(* CODESYS project Monarco HAT library for codesys 0.9.0.3.library
   Author: Aliazzz
   LibDocContent: CommentsAndDocs
   Description: .. _description: 
      
      Library containing device support for Monarco HAT hardware developped by the guys from Monarco.io.
      
      I decided to write this library because the hardware is very solid, but a CODESYS implementation was missing.
      Writing this library was fun, but took a lot of sweat and time, please refer to this work when you use it =).
      
      I am not affiliated with Monarco.io in any way, shape or form.
      
      Released under Unlicense.
      
      
      Enjoy!
      
      
      **Getting started**
      
      To use the HAT, RS-485 and the Realtime Clock under CODESYS, please follow these steps. RTC requires no Linux side config apart from the overlay;
      
      1) On your Raspberry Pi, switch to root user: sudo -s
      
      2) Disable Linux console on UART: **sed 's/ console=serial0,[0-9]\+//' -i /boot/cmdline.txt**
      
      3) Run the following command to get device-tree overlay definition for the RS-485 on the Monarco HAT: **wget www.monarco.io/download/monarco-fix-4-9.dtbo**
      
      4) Copy it to /boot/overlays: **sudo cp monarco-fix-4-9.dtbo /boot/overlays**
      
      5) Afterwards add dtoverlay=monarco-fix-4-9 line to the /boot/config.txt file: **echo dtoverlay=monarco-fix-4-9 >> /boot/config.txt**
      
      6) Reboot your Raspberry Pi: **reboot**
      
      7) After reboot, check the output of the following command: **ls -l /dev/serial0**
      
      8) The response should read **"/dev/serial0 -> ttyAMA0"**
      
      9) Again, switch to root user: **sudo -s  cd etc/**
      
      10) Then: **nano CODESYSControl.cfg**
      
      11) Add the following lines: **[SysCom] Linux.Devicefile=/dev/ttyAMA**
      
      12) Then reboot your Raspberry Pi again: **reboot**
      
      13) After reboot: **Now you can use the HAT, RS-485 and the Real-Time Clock in CODESYS!** from within an IEC application via a comlib of you own flavour (like CAA SerialCOM library).
      
      .. image:: ../Images/MonarcoHAT.png
      
      
      * Real Time Clock (RTC)
      * RS-485 Interface
      * 1-Wire Interface (1w)
      * 4 Digital Inputs
      * 4 Digital Outputs
      * 2 Analog Inputs 12 bits without sign: (0 - 4095) 0..10V / 0..25mA
      * 2 Analog Outputs 12 bit without sign: (0 - 4095) 0..10V
      * LEDs: 1 × orange, 8 × green LEDs
      * Power supply: 10-30 VDC, powers also the Raspberry Pi
      
      
      This library is based on Hardware version 0106, Firmware version 2006.
   Title: Monarco HAT library for Codesys
   Version: 0.9.0.3
   DefaultNamespace: MNR
   DocFormat: reStructuredText
   Company: Monarco.io

Project tree, tasks and I/O mapping:
  libraries: IoDrvGPIO, 3.5.11.0 (3S - Smart Software Solutions GmbH); Raspberry Pi Peripherals, 3.5.11.0 (3S - Smart Software Solutions GmbH); IoStandard, * (System); CAA Memory, * (CAA Technical Workgroup); Standard, * (System); CAA Real Time Clock Extern, * (CAA Technical Workgroup); CAA SerialCom, * (CAA Technical Workgroup)
  function block Monarco_FB [ST]: AfterReadInputs, BeforeWriteOutputs, Initialize, flush, checkCRC, dataTransfer, getCRC, writeRaw, getHATinfo, RS485Baudrate, RS485Mode, HostBaudrate, RS485RxC, RS485TxC, RS485FxC, RS485PxC, setDOut, ServiceRequest, getCpuID, getFwVersion, getHwVersion, getStatus, HWConfig1, Watchdog, getServiceResponse, ControlByte, getDIn, getAIn, setRawTxBuf, getRawRxBuf, setAOut, Counter1Config, Counter2Config, setPWM1freq, setPWM2freq, setDutyCycleDOut1, setDutyCycleDOut2, setDutyCycleDOut3, setDutyCycleDOut4, SetUserLED
  00000000-0000-0000-0000-000000000000|C:\Users\user\Desktop\Monarco HAT\Dev\images\schematics.png
  Library Information/
    function GetLibVersionNumber [ST]
    function GetLibVersion [ST]
    function IsLibReleased [ST]
  Images/
    schematics
    MonarcoHAT
  00000000-0000-0000-0000-000000000000|C:\Users\user\Desktop\Monarco HAT\Dev\images\MonarcoHAT.png
  Datatypes/
    RS485/
      data type stRS485Mode
      data type eRS485Parity
      data type eRS485Databits
      data type eRS485Stopbits
    AIn/
      data type stAIn
    AOut/
      data type stAOut
    DIn/
      data type stDIn
    DOut/
      data type stDOut
    Service/
      data type stServiceRequest
      data type eMonarcoOperation
      data type stMonarcoStatus
      data type eMonarcoComStatus
      data type stMonarcoCmd
      data type stHWConfig1
      data type stControlByte
      data type stHATinfo
      data type eServiceCommand
      data type stServiceResponse
    Counter/
      data type stCounter1Config
      data type eCounterMode
      data type eCounterDirection
      data type eCounterActiveEdge
      data type stCounter2Config
      data type eCounterCapture
    PWM/
      data type ePrescaler
      data type stPWM2
      data type stPWM1
  global variables ParamList
  Functions/
    function getDC [ST]
*)

// Datatypes/Service/stServiceRequest
// Service Request and Service Response structure
// **Setting "Error" is only valid in a Service Response**
TYPE stServiceRequest :
STRUCT
	wServiceValue 	: WORD;
	wServiceAddress : WORD;
/// Error to be examined on a response only! 
/// If set, the response ServiceValue contains one of the following error codes;
///
/// - Invalid adress (code 16#FFFF)
/// 
/// - CRC error (16#CCCC)
///
	xError			: BOOL; 	
END_STRUCT
END_TYPE

// Datatypes/Service/eMonarcoOperation
/// Execution commands for the Monarco HAT via classic command interface
{attribute 'qualified_only'}
{attribute 'strict'}
TYPE eMonarcoOperation :
(
/// Write an entire raw self defined message according to input 
	WriteRaw			:= 0,
/// Write the controlbyte according to input  	
	WriteCtrlByte		:= 1,
/// Write the leds according to input  	
	WriteUserLeds		:= 2,
/// Write Digital Outs according to input	
	WriteDOut			:= 3,
/// Write Analog Outs according to input	
	WriteAOut			:= 4,
/// Write PWM1 frequency according to input	
	WritePWM1Freq		:= 5,
/// Write PWM2 frequency according to input	
	WritePWM2Freq		:= 6,
/// Write Counter1 according to input	
	WriteCNT1			:= 7,
/// Write Counter2 according to input	
	WriteCNT2			:= 8,
/// Write PWM1 duty cycle according to input	
	WriteDutyCycleDOut1	:= 9,
/// Write PWM1 duty cycle according to input	
	WriteDutyCycleDOut2	:= 10,
/// Write PWM1 duty cycle according to input	
	WriteDutyCycleDOut3	:= 11,
/// Write PWM2 duty cycle according to input	
	WriteDutyCycleDOut4	:= 12
) UINT;
END_TYPE

// Datatypes/Service/stMonarcoStatus
/// Monarco HAT Classic Status Structure
{attribute 'qualified_only'}
{attribute 'strict'}
TYPE stMonarcoStatus :
STRUCT
/// Is the Monarco HAT operational?
	xOperational			: BOOL;
/// Operation Command was successfully finished 			 	
	xDone					: BOOL;
/// An errror occuried, see ComStatus			 	
	xError					: BOOL;
/// Has to examined in conjunction with xExecute, xDone and xError				 	
	eComStatus				: eMonarcoComStatus;
/// Controlbyte status 	
	stControlByte			: stControlByte; 
/// Contains most recent service response	
	stLastServiceResponse	: stServiceResponse;
/// User Leds On Off status;
	byUserLeds				:BYTE;
/// Current state of digital In channel values  	
	stDIn					: stDIn;
/// copy of digital Out channel values				
	stDOut					: stDOut;
/// Current state of analog In channel values  				
	stAIn					: stAIn;
/// copy of analog Out channel values
	stAOut					: stAOut;
/// current watchdog time: 100 = 100msec
	uiWatchDog				: UINT;
/// current Baudrate: 300 = 300Bd				
	uiRS485Baudrate			: UINT;
/// Current RS485 communication settings mode				
	stRS485Mode				: stRS485Mode;
/// Current settings for RS485 termination and AI voltage or current-loop mode			
	stHWConfig1 			: stHWConfig1;
/// Current Counter 1 configuration  			
	stCounter1Config		: stCounter1Config;
/// Current Counter 2 configuration	
	stCounter2Config		: stCounter2Config;
/// PWM1 Settings
	stPWM1					: stPWM1;
/// PWM2 Setting
	stPWM2					: stPWM2;
/// Static HAT information like FW version, HW version and CPU ID 	
	stHATinfo				: stHATinfo;
/// RAW receive buffer			
	abyRawRxBuffer			: ARRAY [0..(ParamList.MONARCO_STRUCT_SIZE-1)] OF BYTE; 
END_STRUCT
END_TYPE

// Datatypes/Service/eMonarcoComStatus
/// Monarco HAT Communication Status
{attribute 'qualified_only'}
{attribute 'strict'}
TYPE eMonarcoComStatus :
(	
/// Succes: Rx/Tx sent succesfully
	Succes			 		:= 0,
/// Error: Rx/Tx fail
	Error					:= 1,
/// Device not found on the bus
	SPIdeviceNotFound		:= 2,
/// No commands are currently executed. Is xExecute command on the Function Block set?
	SPIidleNoExecute		:= 3,
/// The received message was crippled and dropped
	CrcFail 				:= 4 
) UINT;
END_TYPE

// Datatypes/Service/stMonarcoCmd
/// Monarco Classic Command Structure
{attribute 'qualified_only'}
{attribute 'strict'}
TYPE stMonarcoCmd :
STRUCT
/// Starts a single operation of type "eFunction" on a rising edge of xExecute
	xExecute			: BOOL;	
/// Command to be executed on rising edge of "xExecute"			
	eOperation			: eMonarcoOperation;
/// Use in combination with "eOperation.WRITE_RAW". Setting a CRC is not neccesary, it will be calculated and added automatically	
	abyTxBuffer			: ARRAY [0..(ParamList.MONARCO_STRUCT_SIZE-1)] OF BYTE;
/// For use in combination with "eOperation.WRITE_CTRLBYTE"
	stControlByte		: stControlByte;
/// For use in combination with "eOperation.WRITE_USERLEDS"
	byLeds				: BYTE;
/// For use in combination with "eOperation.WRITE_DOut"		
	stDOut				: stDOUT;
/// For use in combination with "eOperation.WRITE_AOut"			
	stAOut				: stAOut;
/// For use in combination with "eOperation.WRITE_Counter1"			
	stCounter1			: stCounter1Config;
/// For use in combination with "eOperation.WRITE_Counter2"
	stCounter2			: stCounter2Config;
/// For use in combination with "eOperation.WRITE_PWM1Frequency" 
	PWM1freq			: UDINT;
/// For use in combination with "eOperation.WRITE_PWM2Frequency" 
	PWM2freq			: UDINT;
/// For use in combination with "eOperation.WRITE_DutyCycleDOut1" 
	rDutyCycleDOut1		: REAL;
/// For use in combination with "eOperation.WRITE_DutyCycleDOut1" 
	rDutyCycleDOut2		: REAL;
/// For use in combination with "eOperation.WRITE_DutyCycleDOut1" 
	rDutyCycleDOut3		: REAL;
/// For use in combination with "eOperation.WRITE_DutyCycleDOut1" 
	rDutyCycleDOut4		: REAL;
END_STRUCT
END_TYPE

// Datatypes/Service/stHWConfig1
/// Set AnalogIn Channels to Voltage or Current Loop mode,
/// Set RS-485 termination resistor
TYPE stHWConfig1 :
STRUCT
/// AIN1 current loop shunt resistor enable (TRUE / FALSE)
    xAIn1shunt  	: BOOL; 
/// AIN2 current loop shunt resistor enable (TRUE / FALSE)
    xAIn2shunt  	: BOOL;
/// RS-485 termination resistor enable (TRUE / FALSE)
	xTerminated		: BOOL;	
END_STRUCT
END_TYPE

// Datatypes/AOut/stAOut
/// Analog Outputs
TYPE stAOut :
STRUCT
	/// 0..4095 = 0..10V
	wAOut1			: WORD;
	/// 0..4095 = 0..10V
	wAOut2			: WORD; 
END_STRUCT
END_TYPE

// Datatypes/Service/stControlByte
TYPE stControlByte :
STRUCT
/// Status LED mask
/// set 1 for control LED0 by Control byte / Status LED on
/// set 0 for default LED0 function (system status indication, see Monarco HAT Hardware Reference Manual)
	xStatusLedCtrl		: BOOL;
/// Status LED on 
/// Set 1 for LED0 lit on 
/// Set 0 for LED0 off: only applicable if Control byte / Status LED mask set 1
	xStatusLedValue		: BOOL;
/// 1-Wire power shutdown 
/// Set 1 for 1-Wire bus power down (useful for bus reset in case of freeze) 
/// Set 0 for normal operation
	xOneWireShutdown	: BOOL;
/// RESERVED - allways set 0
	xReserved 			: BOOL := FALSE;
/// Counter 1 reset 
/// Set 1 for COUNTER1 Value reset request
/// Set 0 for normal operation. 
/// Reset operation is edge-triggered and its completion is signalised by Statusbyte/Counter 1/2 reset done bit
	xCounter1Reset		: BOOL;
/// Counter 2 reset 
/// Set 1 for COUNTER2 Value reset request
/// Set 0 for normal operation. 
/// Reset operation is edge-triggered and its completion is signalised by Statusbyte/Counter 1/2 reset done bit
	xCounter2Reset		: BOOL;
/// [FUTURE] Sign of Life 0/1 - should be incremented with each data transfer as 2bit number low/high bit, used by firmware as health check of SPI Master
	xSignOfLife0		: BOOL;
/// [FUTURE] Sign of Life 0/1 - should be incremented with each data transfer as 2bit number low/high bit, used by firmware as health check of SPI Master
	xSignOfLife1		: BOOL; 
END_STRUCT
END_TYPE

// Datatypes/DIn/stDIn
/// Digital Inputs
TYPE stDIn :
STRUCT
	xDIn1			: BOOL;
	xDIn2			: BOOL;
	xDIn3			: BOOL;
	xDIn4			: BOOL;
END_STRUCT
END_TYPE

// Datatypes/Service/stHATinfo
/// Returns Firmware, Hardware and CPU revision
TYPE stHATinfo :
STRUCT
/// Monarco HAT Firmware Version
	dwFwVersion			: DWORD;
/// Monarco HAT Hardware Version 
	dwHwversion			: DWORD;
/// Monarco HAT MCU CPU ID
	lwCpuID				: LWORD;
END_STRUCT
END_TYPE

// Datatypes/AIn/stAIn
/// Analog Inputs
TYPE stAIn :
STRUCT
	/// 0..4095 equals 0..10V or 0..25mA, see stHWConfig1_
	wAIn1			: WORD;
	/// 0..4095 equals 0..10V or 0..25mA, see stHWConfig1_
	wAIn2			: WORD;
END_STRUCT
END_TYPE

// Datatypes/DOut/stDOut
/// Digital Outputs
TYPE stDOut :
STRUCT
	xDOut1				: BOOL;
	xDOut2				: BOOL; 
	xDOut3				: BOOL;
	xDOut4				: BOOL; 
END_STRUCT
END_TYPE

// Datatypes/Service/eServiceCommand
/// Registers are Read-only [R], Read-Write [RW] or Write-only [W].
{attribute 'qualified_only'}
{attribute 'strict'}
TYPE eServiceCommand  :
(
/// Read: 0xABCD = OK, [FUTURE] "watchdog triggered", 
/// Write [FUTURE]: - accept only 0xABCD = reset status
	SDC_FIXED_STATUSWORD := 16#0000,
/// Firmware Version - Low Word [R] 
	SDC_FIXED_FWVERL	 := 16#0001,
/// Firmware Version - High Word [R] 
	SDC_FIXED_FWVERH	 := 16#0002,
/// Hardware Version - Low Word [R]
	SDC_FIXED_HWVERL	 := 16#0003,
/// Hardware Version - High Word [R]
	SDC_FIXED_HWVERH	 := 16#0004,
/// MCU Unique ID 1 [R]
	SDC_FIXED_CPUID1	 := 16#0005, 
/// MCU Unique ID 2 [R]
	SDC_FIXED_CPUID2	 := 16#0006, 
/// MCU Unique ID 3 [R]
	SDC_FIXED_CPUID3	 := 16#0007,
/// MCU Unique ID 4 [R]
	SDC_FIXED_CPUID4	 := 16#0008, 
/// HW Config 1 [RW]
/// 
/// * bit 00 - RS-485 termination resistor enable
/// 
/// * bit 01 - AIN1 current loop shunt resistor enable
///  
/// * bit 02 - AIN2 current loop shunt resistor enable
/// 
/// * bit 03..15 - RESERVED (write zeros)
	SDC_FIXED_HWConfig1  := 16#000A,
/// Watchdog Timeout [RW]
/// 
/// Unit: 1 ms; 0 = watchdog disabled; default = 100
	SDC_FIXED_WATCHDOG	 := 16#000F, 
/// HAT RS-485 Baudrate [RW]
///  
/// Unit: 100 Bd, Min: 3 (300 Bd), Max 10000 (1 MBd)
	SDC_FIXED_RS485BAUD  := 16#0010, 
/// HAT RS-485 Mode [RW]
/// 
/// * bit 00..02 - parity - 0: none, 1: even, 2: odd;
/// 
/// * bit 03..04 - data bits: 0: 5, 1: 6, 2: 7, 3: 8; 
/// 
/// * bit 05..06 - stop bits: 0: half, 1: one, 2: one and half, 3: two; 
/// 
/// * bit 07..15 - RESERVED (write zeros)
	SDC_FIXED_RS485MODE  := 16#0011,
/// Host (Pi) UART Baudrate [RW] Unit: 100 Bd, Min: 3 (300 Bd), Max 10000 (1 MBd); 
/// 
/// set to 0 to disable Host UART (set Monarco pins to Hi-Z) when you are using it for another external device.
	SDC_FIXED_HOST_UART  := 16#0012,
/// RS-485 Bytes Received Diagnostics Counter [R]
	SDC_FIXED_RS485_RxC	 := 16#0014,
/// RS-485 Bytes Transmitted Diagnostics Counter [R]
    SDC_FIXED_RS485_TxC  := 16#0015,
/// RS-485 RX Framing Error Diagnostics Counter [R]
    SDC_FIXED_RS485_FxC	 := 16#0018,
/// RS-485 RX Parity Error Diagnostics Counter [R]
    SDC_FIXED_RS485_PxC  := 16#0019,
/// COUNTER1 Configuration [W]
/// 
/// * bit 00..02 - mode: 0: off, 1: pulse counting, 2: quadrature encoder,
/// 
/// * bit 03..05 - direction (only for pulse counting mode): 0: up, 1: [FUTURE] external control, low/high = up/down,
/// 
/// * bit 06..07 - active edge (only for pulse counting mode): 0: rising, 1: falling, 2: both,
/// 
/// * bit 08..15 - RESERVED (write zeros)
	SDC_FIXED_CNT1MODE 	 := 16#0024, 
/// COUNTER2 Configuration [W]
/// 
/// * bit 00..02 - mode: 0: off, 1: pulse counting, 2: quadrature encoder,
/// 
/// * bit 03..05 - direction (only for pulse counting mode): 0: up, 1: [FUTURE] external control, low/high = up/down,
/// 
/// * bit 06..07 - active edge (only for pulse counting mode): 0: rising, 1: falling, 2: both,
/// 
/// * bit 08..09 - CAPTURE function active edge: 0: disabled, 2: [FUTURE] falling, 3: [FUTURE] both,
/// 
/// * bit 10..15 - RESERVED (write zeros)
	SDC_FIXED_CNT2MODE	 := 16#0025,
/// PERSISTENT [FUTURE] parameters area (64 registers, 128 BYTE) 
/// Now for manufacturer use only.
	SDC_PERSISTENT_MIN 	 := 16#0F00,
/// PERSISTENT [FUTURE] parameters area (64 registers, 128 BYTE) 
/// Now for manufacturer use only. 
	SDC_PERSISTENT_MAX 	 := 16#0F3F  
) UINT;
END_TYPE

// Datatypes/RS485/stRS485Mode
/// Monarco HAT RS485 UART settings
TYPE stRS485Mode :
STRUCT
	eParity		 : eRS485Parity;
	eDatabits	 : eRS485Databits;
	eStopbits	 : eRS485Stopbits;
END_STRUCT
END_TYPE

// Datatypes/RS485/eRS485Parity
{attribute 'qualified_only'}
{attribute 'strict'}
TYPE eRS485Parity :
(
	None := 0, 	/// No parity check
	Even := 1,	/// Even parity check
 	Odd  := 2	/// Odd parity check
) UINT;
END_TYPE

// Datatypes/RS485/eRS485Databits
{attribute 'qualified_only'}
{attribute 'strict'}
TYPE eRS485Databits :
(
	Five 	:= 0,	// 1 Byte contains 5 databits
	Six 	:= 1,	// 1 Byte contains 6 databits
	Seven 	:= 2,	// 1 Byte contains 7 databits
	Eight 	:= 3	// 1 Byte contains 8 databits
) UINT;
END_TYPE

// Datatypes/RS485/eRS485Stopbits
{attribute 'qualified_only'}
{attribute 'strict'}
TYPE eRS485Stopbits :
(
	Half 		:= 0,	// 1/2 stopbit
	One 		:= 1,	// 1 stopbit
	OneAndAHalf := 2,	// 1-1/2 stopbits
	Two 		:= 3	// 2 stopbits
) UINT;
END_TYPE

// Datatypes/Service/stServiceResponse
// Alias of Service Request
TYPE stServiceResponse : stServiceRequest; 
END_TYPE

// Datatypes/Counter/stCounter1Config
/// COUNTER1 Configuration;
///   Mode;
///	   * Off,
///    * Pulse counting,
///    * Quadrature encoder,
///   Direction (only for pulse counting mode):
///     * Up
///     * [FUTURE] external control, low/high = up/down
///   Active Edge (only for pulse counting mode):
///     * Rising
///     * Falling
///     * Both
TYPE stCounter1Config :
STRUCT
	eMode		: eCounterMode;
	eDirection	: eCounterDirection;
	eActiveEdge	: eCounterActiveEdge;
END_STRUCT
END_TYPE

// Datatypes/Counter/eCounterMode
{attribute 'qualified_only'}
{attribute 'strict'}
TYPE eCounterMode :
(
	Off 				:= 0,
	PulseCounting		:= 1,
	QuadratureEncoder	:= 2
) UINT;
END_TYPE

// Datatypes/Counter/eCounterDirection
{attribute 'qualified_only'}
{attribute 'strict'}
TYPE eCounterDirection :
(
	Up					:= 0,
	External_Control1	:= 1 //[FUTURE] external control, low/high = up/down
) UINT;
END_TYPE

// Datatypes/Counter/eCounterActiveEdge
{attribute 'qualified_only'}
{attribute 'strict'}
TYPE eCounterActiveEdge :
(
	Rising	:= 0,
	Falling	:= 1,
	Both	:= 2
) UINT;
END_TYPE

// Datatypes/Counter/stCounter2Config
/// COUNTER2 Configuration;
///   Mode;
///	   * Off,
///    * Pulse counting,
///    * Quadrature encoder,
///   Direction (only for pulse counting mode):
///     * Up
///     * [FUTURE] external control, low/high = up/down
///   Active Edge (only for pulse counting mode):
///     * Rising
///     * Falling
///     * Both
///   CAPTURE function active edge:
///     * Disabled
///     * [FUTURE] rising
///     * [FUTURE] falling
///     * [FUTURE] both
TYPE stCounter2Config : 
STRUCT
	Mode		: eCounterMode;
	Direction	: eCounterDirection;
	ActiveEdge	: eCounterActiveEdge;
	Capture		: eCounterCapture;
END_STRUCT
END_TYPE;

// Datatypes/Counter/eCounterCapture
{attribute 'qualified_only'}
{attribute 'strict'}
TYPE eCounterCapture :
(
	Disabled 	:= 0,
	Rising 		:= 1, // [FUTURE]
	Falling 	:= 2, // [FUTURE]
	Both		:= 3  // [FUTURE]
) UINT;
END_TYPE

// Datatypes/PWM/ePrescaler
{attribute 'qualified_only'}
{attribute 'strict'}
TYPE ePrescaler :
(	
	ScaleFactor1	:= 0,	/// PWM Prescale factor is set to 1
	ScaleFactor8 	:= 1,	/// PWM Prescale factor is set to 8
	ScaleFactor64 	:= 2,	/// PWM Prescale factor is set to 64
	ScaleFactor512 	:= 3	/// PWM Prescale factor is set to 512
) UDINT;
END_TYPE

// Datatypes/PWM/stPWM2
TYPE stPWM2 :
STRUCT
	/// period of PWM2 Ch A (DOut4)	(Hz)
	Freq			: UDINT;
	/// Duty Cycle of PWM2 Ch A (DOut4)	
	DutyCycleDOut4	: REAL;
END_STRUCT
END_TYPE

// Datatypes/PWM/stPWM1
TYPE stPWM1 :
STRUCT
	/// period of PWM1 Ch A, B and C (DOut1, 2 and 3) (Hz)
	Freq			: UDINT;
	/// Duty Cycle of PWM1 Ch A (DOut1)	
	DutyCycleDOut1	: REAL;
	/// Duty Cycle of PWM1 Ch B (DOut2)	
	DutyCycleDOut2	: REAL;
	/// Duty Cycle of PWM1 Ch C (DOut3)	
	DutyCycleDOut3	: REAL;
END_STRUCT
END_TYPE

// ParamList
{attribute 'qualified_only'}
VAR_GLOBAL CONSTANT
	MONARCO_STRUCT_SIZE 				: UINT := 26;	
	MONARCO_SERVICE_STATUS_OK 			: WORD := 16#ABCD;
	MONARCO_SERVICE_ERROR_UNKNOWN_REG 	: WORD := 16#FFFF;
	MONARCO_SERVICE_ERROR_CRC 			: WORD := 16#CCCC;
	SDC_ADDRESS_MASK					: WORD := 16#0FFF;		                            
	MONARCO_ADC_RANGE_MAX 				: WORD := 16#4095;
END_VAR

// Monarco_FB
FUNCTION_BLOCK Monarco_FB EXTENDS SPI
VAR_INPUT
	Cmd						: stMonarcoCmd;
END_VAR
VAR_OUTPUT
	Status					: stMonarcoStatus;
END_VAR
VAR
	uiNumberOfDevices		: UINT;		/// Beware, this Library does **NOT** support implementation of multiple SPI devices!
	xGetInitialStatusInfo	: BOOL;		/// Get status info on startup once
	fbR_TRIG				: R_TRIG;	/// FB internal rising edge trigger for xExecute input
	abyIntTxBuf				: ARRAY [0..(ParamList.MONARCO_STRUCT_SIZE-1)] OF BYTE;  
	abyIntRxBuf				: ARRAY [0..(ParamList.MONARCO_STRUCT_SIZE-1)] OF BYTE;  
END_VAR

//********************************
//	base SPI implementation 
//********************************
SUPER^();


//********************************
//		get SPI State 
//********************************
CASE _iState OF
0:
	IF SUPER^.init() THEN
		_iState := 1;
	END_IF	

1:	
	_iState := 10;
	xGetInitialStatusInfo := TRUE;
END_CASE


//********************************
//		is device operational 
//********************************
IF _iState = 10 THEN
	Status.xOperational		:=	TRUE;
ELSE
	Status.xOperational		:=	FALSE;
END_IF


//********************************
// Get Initial startup Status Info 
//******************************** 
IF xGetInitialStatusInfo THEN
	THIS^.getHATinfo();				// all property calls are done via status.gthatinfo to reduce SPI bandwidth on ponintless static info.
	THIS^.Status.stControlByte		:= THIS^.ControlByte;	
	THIS^.Status.stHWConfig1		:= THIS^.HWConfig1;
	THIS^.Status.uiRS485Baudrate	:= THIS^.RS485Baudrate;
	THIS^.Status.stRS485Mode	 	:= THIS^.RS485Mode;
	THIS^.Status.uiWatchDog		 	:= THIS^.Watchdog;
	THIS^.Status.stCounter1Config	:= THIS^.Counter1Config;
	THIS^.Status.stCounter2Config	:= THIS^.Counter2Config;	
	xGetInitialStatusInfo 			:= FALSE;
END_IF


//********************************
//		Operation Mode
//********************************
// No execute, set feedback to inform user
IF NOT Cmd.xExecute THEN				
	Status.xError			:=	FALSE;
	Status.xDone			:=  FALSE;
	Status.eComStatus		:= 	eMonarcoComStatus.SPIIdleNoExecute;
END_IF


fbR_TRIG(CLK:= Cmd.xExecute);

IF fbR_TRIG.Q THEN
	
	CASE Cmd.eOperation	OF
		///********************************
		///	 Add classic operations here
		///********************************
		eMonarcoOperation.WriteRaw				:	Status.eComStatus 		:= THIS^.writeRaw();
		eMonarcoOperation.WriteCtrlByte			: 	THIS^.ControlByte		:= CMD.stControlByte;
		eMonarcoOperation.WriteUserLeds			:   Status.eComStatus		:= THIS^.SetUserLED(byLeds := Cmd.byLeds);
		eMonarcoOperation.WriteDOut				: 	Status.eComStatus 		:= THIS^.setDOut(stDOut := CMD.stDOut);
		eMonarcoOperation.WriteAOut				: 	Status.eComStatus 		:= THIS^.setAout(stAOut := CMD.stAOut);
		eMonarcoOperation.WriteCNT1				: 	THIS^.Counter1Config	:= Cmd.stCounter1;
		eMonarcoOperation.WriteCNT2				: 	THIS^.Counter2Config 	:= Cmd.stCounter2;                 	
		eMonarcoOperation.WritePWM1Freq			: 	Status.eComStatus		:= THIS^.setPWM1freq(udiHz := CMD.PWM1freq);
		eMonarcoOperation.WritePWM2Freq			: 	Status.eComStatus		:= THIS^.setPWM2freq(udiHz := CMD.PWM2freq);
		eMonarcoOperation.WriteDutyCycleDOut1	:	Status.eComStatus		:= THIS^.setDutyCycleDOut1(rDutyCycle := CMD.rDutyCycleDOut1 );
		eMonarcoOperation.WriteDutyCycleDOut2	:	Status.eComStatus		:= THIS^.setDutyCycleDOut1(rDutyCycle := CMD.rDutyCycleDOut2 );	
		eMonarcoOperation.WriteDutyCycleDOut3	:	Status.eComStatus		:= THIS^.setDutyCycleDOut1(rDutyCycle := CMD.rDutyCycleDOut3 );	
		eMonarcoOperation.WriteDutyCycleDOut4	:	Status.eComStatus		:= THIS^.setDutyCycleDOut2(rDutyCycle := CMD.rDutyCycleDOut4 );	
	END_CASE 

	IF status.eComStatus = eMonarcoComStatus.SUCCES THEN 			
		Status.xDone			:= TRUE;
		Status.abyRawRxBuffer	:= abyIntRxBuf;
	ELSE
		Status.xError			:= TRUE;
	END_IF

END_IF

METHOD AfterReadInputs : INT
VAR
	aby: ARRAY[0..2] OF BYTE;	
	usiChannel: USINT;
	ui: UINT;
END_VAR
SUPER^.AfterReadInputs();
END_METHOD

METHOD BeforeWriteOutputs : INT
VAR
	i: USINT;
END_VAR
SUPER^.BeforeWriteOutputs();
END_METHOD

METHOD Initialize   : UDINT
VAR_INPUT
	wModuleType     : UINT;
	dwInstance      : UDINT;
	pConnector      : POINTER TO IoConfigConnector;
END_VAR
VAR
	pParam			: POINTER TO IoConfigParameter;	
	pParam1			: POINTER TO DWORD;	
	udiResult		: UDINT;
	i				: INT;
END_VAR
SUPER^.Initialize(wModuleType, dwInstance, pConnector);


//********************************
//	 Set the number of devices 
//********************************
pParam := ConfigGetParameter(_pConnector, 1);

IF pParam <> 0 THEN
	THIS^.uiNumberOfDevices := IoStandard.ConfigGetParameterValueByte(pParam, ADR(udiResult));
END_IF


//********************************
//	 Set parameters of devices 
//********************************
FOR i := 0 TO UINT_TO_INT(THIS^.uiNumberOfDevices - 1) DO
	pParam 			:= ConfigGetParameter(_pConnector, 100 + INT_TO_UINT(i));
	pParam1			:= IoStandard.ConfigGetParameterValuePointer(pParam, ADR(udiResult));
END_FOR;
END_METHOD

// Initialises the entire buffer with 16#00 (flush)
METHOD PRIVATE flush : BOOL
VAR_INPUT
	abyRxBuf			: ARRAY [0..(ParamList.MONARCO_STRUCT_SIZE-1)] OF BYTE;
END_VAR
VAR
	i				: UINT;
END_VAR
//flush the temporary receive buffer before filling;
FOR i :=0 TO (ParamList.MONARCO_STRUCT_SIZE-1) DO
	abyRxBuf[i] := 16#00;
END_FOR
flush := TRUE;
END_METHOD

METHOD PRIVATE checkCRC : BOOL
VAR_INPUT
	abyRxBuf		: ARRAY [0..(ParamList.MONARCO_STRUCT_SIZE-1)] OF BYTE;
END_VAR
VAR
	CRC				: WORD;
	CRCLo			: BYTE;
	CRCHi			: BYTE;
END_VAR
CRC 			:= THIS^.GetCRC(abyRxBuf);
CRCHi			:= WORD_TO_BYTE(CRC);
CRCLo 			:= WORD_TO_BYTE(SHR(CRC,8));

// check to self calculated CRC against the sent CRC, Equal = OK
IF (CRCHi = abyRxBuf[ParamList.MONARCO_STRUCT_SIZE - 2]) AND (CRCLo = abyRxBuf[ParamList.MONARCO_STRUCT_SIZE - 1]) THEN 
	checkCRC := TRUE;
ELSE
	checkCRC := FALSE;
END_IF;
END_METHOD

(* Handles the SPI data transfer to the Monarco Hat *)
METHOD PRIVATE dataTransfer 	: eMonarcoComStatus
VAR                 	
	tmpRxBuf			: ARRAY [0..(ParamList.MONARCO_STRUCT_SIZE-1)] OF BYTE;  
	udiBufSize			: UDINT;          
	xDone				: BOOL;
	CRC					: WORD;
END_VAR
//init temporay buffer before filling;
//flush(tmpRxBuf);

// determine size of buffer
udiBufSize 						:= SIZEOF( THIS^.abyIntTxBuf );

(* Sets CRC16 checksum, for Tx byte array [24] and [25]*)
CRC 							:= THIS^.getCRC( THIS^.abyIntTxBuf );
THIS^.abyIntTxBuf[24]			:= WORD_TO_BYTE(CRC);
THIS^.abyIntTxBuf[25]			:= WORD_TO_BYTE(SHR(CRC,8));

// Send, Recv
xDone := THIS^.transferExt( pabyTxBuffer := ADR( THIS^.abyIntTxBuf ), 
						 pabyRxBuffer := ADR( tmpRxBuf ), 		// write result into a temporary buffer for post-analysis. Beware that the received answser is from the last question, not the current question.
						 udiLen		  := udiBufSize, 
						 uiDelayus	  := 5,
						 udispeedHz	  := 0); 

IF NOT xDone THEN 
	// Send, Recv failed
	DataTransfer := eMonarcoComStatus.ERROR;
ELSE
	// OK?
	IF THIS^.checkCRC(tmpRxBuf) THEN
		//CRC okay, return the recv buffer
		THIS^.abyIntRxBuf 	:= tmpRxBuf;
		DataTransfer		:= eMonarcoComStatus.SUCCES;
	ELSE
		//CRC not okay, return an empty buffer
		flush(tmpRxBuf);
		THIS^.abyIntRxBuf 	:= tmpRxBuf;
		DataTransfer		:= eMonarcoComStatus.CrcFail;
	END_IF
END_IF;
END_METHOD

//Returns CRC16 checksum for input buffer
//byte 24 and 25 are not taken in account, they hold the crc16 itself
METHOD PRIVATE getCRC : WORD
VAR_INPUT
	abyBuf			: ARRAY [0..(ParamList.MONARCO_STRUCT_SIZE-1)] OF BYTE;
END_VAR
VAR
	uiSizeTx 		: UINT;
	udiCRCLen 		: UDINT;
	pByteTx  		: POINTER TO BYTE;
	CheckSum		: WORD; 
END_VAR
// startadress of bytes
pByteTx								:= ADR(abyBuf); 

// calculate CRC-16 checksum, beware that for the checksum calculation, we need to skip the checksum itself
uiSizeTx							:= SIZEOF(abyBuf);

// should always be 24 / 16#18
udiCRCLen							:= (uiSizeTx -16#02);	
	
CheckSum							:= MEM.CRC16_Modbus( pByteTx, TO_UINT(udiCRCLen) );

// return checksum
getCRC 								:= CheckSum;
END_METHOD

// Set a RAW buffer
METHOD PRIVATE writeRaw : eMonarcoComStatus
VAR
	CRC	: WORD;
END_VAR
//Copy the cmd buffer to internal buffer
abyIntTxBuf 					:= Cmd.abyTxBuffer;

//Sets CRC16 checksum, for Tx byte array [24] and [25]
CRC 							:= THIS^.getCRC( THIS^.abyIntTxBuf );

// word -> word_to_byte -> highbyte (C6)
THIS^.abyIntTxBuf[24]			:= WORD_TO_BYTE(CRC);
	
// word -> word_to_byte([shr] 8 bits) -> lowbyte (E1)
THIS^.abyIntTxBuf[25]			:= WORD_TO_BYTE(SHR(CRC,8));

//send/receive
WriteRaw 						:= THIS^.dataTransfer();
END_METHOD

//Read current FW, HW revision and CPU-ID 		
METHOD PRIVATE getHATinfo
VAR
	wValue				: WORD;
	eCmd				: eServiceCommand;
	J					: INT;
	wReqAdr	 	  		: WORD;
	awSrvAnwser			: ARRAY [1..9] OF WORD;
	cpu_l				: DWORD;
	cpu_h 				: DWORD;
	lwcpu				: LWORD;
END_VAR
//********************************
//Read FW, HW revision and CPU-ID 
//******************************** 
FOR J := 1 TO 9 DO
	CASE J OF
		1:		eCmd := eServiceCommand.SDC_FIXED_FWVERL;
		2:		eCmd := eServiceCommand.SDC_FIXED_FWVERH;
		3:		eCmd := eServiceCommand.SDC_FIXED_HWVERL;
		4:		eCmd := eServiceCommand.SDC_FIXED_HWVERH;
		5:		eCmd := eServiceCommand.SDC_FIXED_CPUID1;
		6:		eCmd := eServiceCommand.SDC_FIXED_CPUID2;
		7:		eCmd := eServiceCommand.SDC_FIXED_CPUID3;
		8:		eCmd := eServiceCommand.SDC_FIXED_CPUID4;
		9:		eCmd := eServiceCommand.SDC_FIXED_STATUSWORD; //bogus question to receive last value (cpuid4)
	END_CASE
	wValue 				:= TO_WORD(eServiceCommand.SDC_FIXED_STATUSWORD);
	Status.eComStatus 	:= THIS^.ServiceRequest( wValue := wValue, eCommand := eCmd, xWrite := FALSE );
	// Get result
	abyIntRxBuf 		:= THIS^.getRawRxBuf();
	awSrvAnwser[J]		:= MEM.PackBytesToWord(abyIntRxBuf[1], abyIntRxBuf[0]);
END_FOR

// Store anwsers in status
Status.stHATinfo.dwFWVersion 		:= MEM.PackWordsToDword(awSrvAnwser[3],awSrvAnwser[2]);
Status.stHATinfo.dwHWversion		:= MEM.PackWordsToDword(awSrvAnwser[5],awSrvAnwser[4]);
cpu_l								:= MEM.PackWordsToDword(awSrvAnwser[7],awSrvAnwser[6]);
cpu_h								:= MEM.PackWordsToDword(awSrvAnwser[9],awSrvAnwser[8]);
lwcpu								:= cpu_h;
lwcpu								:= SHL(lwcpu,32);
status.stHATinfo.lwCpuID			:= lwcpu OR cpu_l;
END_METHOD

/// Please refer to Monarco HAT SPI Protocol Reference Manual for more details!
///
/// Get/Set Monarco HAT RS-485 Baudrate in steps of 100 Baud 
/// 	* Unit: 100 Bd, Min: 3 (300 Bd), Max 10000 (1 MegaBd)
/// 	12 = 1200 Bd, 
/// 	24 = 2400 Bd, 
/// 	48 = 4800 Bd,
/// 	96 = 9600 Bd,
/// 	192 = 19200 Bd, 
/// 	384 = 38400 Bd,
/// 	576 = 57600 Bd,
/// 	1152 = 115200 Bd
PROPERTY RS485Baudrate : UINT
SET
VAR
	uiRate	: UINT;
END_VAR
uiRate := LIMIT( 3, RS485Baudrate, 10000 ); // limit baudrate within accepted range [300 .. 1000000]
Status.eComStatus := THIS^.ServiceRequest( wValue := uiRate, eCommand := eServiceCommand.SDC_FIXED_RS485BAUD, xWrite := TRUE );
END_SET
GET
VAR
	J				 : INT;
	awSrvAnwser		 : ARRAY [1..2] OF WORD;
END_VAR
FOR J := 1 TO 2 DO
	Status.eComStatus 		:= THIS^.ServiceRequest( wValue := 16#0000, eCommand := eServiceCommand.SDC_FIXED_RS485BAUD, xWrite := FALSE  ) ;
	awSrvAnwser[J]			:= MEM.PackBytesToWord(THIS^.abyIntRxBuf[1], THIS^.abyIntRxBuf[0]);
END_FOR

RS485Baudrate 				:= awSrvAnwser[2];

//update classic status
Status.uiRS485Baudrate		:= RS485Baudrate;
END_GET
END_PROPERTY

/// Please refer to Monarco HAT SPI Protocol Reference Manual for more details!
///
/// Read/ Write Host Baudrate in steps of 100 Baud.
/// The host side baudrate is configurable by service register 0x012, but it is usually *NOT* needed, as RS-485 side communication parameters are independant on Host side.
///
/// Default communication parameters on Raspberry Pi (Host side) side are; 
/// 	* 115200 Baud, 
/// 	* 8 data bits, no parity, 
///		* 1 stop Bit/// 115200 Baud, 8 data bits, no parity, 1 stop BIT. 
/// Host side baudrate is configurable by service register 0x012, but it is usually *NOT* needed, 
/// as RS-485 side communication parameters are independant on Host side.
///
/// Monarco HAT RS-485 side communication parameters can be fully configured by service registers 0x010 and 0x011. 
/// Default settings are: 9600 Baud, no parity, 1 stop bit (9k6, 8-N-1). 
///
/// sets RS485 port to
/// * parity - 0: none, 1: even, 2: odd,
/// * data bits: 0: 5, 1: 6, 2: 7, 3: 8,
/// * stop bits: 0: half, 1: one, 2: one and half, 3: two.
PROPERTY RS485Mode : stRS485Mode
SET
VAR
	stMode					: stRS485Mode;
	wReq					: WORD;
END_VAR
//RS-485 Mode [RW]
//  bit 00..02 - parity - 0: none, 1: even, 2: odd
//  bit 03..04 - data bits: 0: 5, 1: 6, 2: 7, 3: 8
//  bit 05..06 - stop bits: 0: half, 1: one, 2: one and half, 3: two
//  bit 07..15 - RESERVED (write zeros)
//
stMode   := RS485Mode;
CASE stMode.eParity OF
	eRS485Parity.none			: 	wReq.0 := FALSE;	//0x00
									wReq.1 := FALSE;
									wReq.2 := FALSE;
									
	eRS485Parity.even 			:  	wReq.0 := TRUE;		//0x01
									wReq.1 := FALSE;
									wReq.2 := FALSE;
									
	eRS485Parity.odd 			:  	wReq.0 := FALSE;	//0x02
									wReq.1 := TRUE;
									wReq.2 := FALSE;
END_CASE

CASE stMode.eDatabits OF
	eRS485Databits.Five 		:  	wReq.3 := FALSE;	//0x00
									wReq.4 := FALSE;
									
	eRS485Databits.Six 			: 	wReq.3 := TRUE;		//0x01
									wReq.4 := FALSE;
									
	eRS485Databits.Seven		:	wReq.3 := FALSE;	//0x02
									wReq.4 := TRUE;
									
	eRS485Databits.Eight		: 	wReq.3 := TRUE;		//0x03
									wReq.4 := TRUE;
END_CASE

CASE stMode.eStopbits OF
	eRS485Stopbits.Half 		:	wReq.5 := FALSE;	//0x00
									wReq.6 := FALSE;
									
	eRS485Stopbits.One  		: 	wReq.5 := TRUE;		//0x01
									wReq.6 := FALSE;
									
	eRS485Stopbits.OneAndAHalf	: 	wReq.5 := FALSE;	//0x02
									wReq.6 := TRUE;
									
	eRS485Stopbits.Two			: 	wReq.5 := TRUE;		//0x03
									wReq.6 := TRUE;
END_CASE

wReq.7 := FALSE;	// Mandatory
wReq.8 := FALSE;	// Mandatory
wReq.9 := FALSE;	// Mandatory
wReq.10 := FALSE;   // Mandatory
wReq.11 := FALSE;   // Mandatory
wReq.12 := FALSE;   // Mandatory
wReq.13 := FALSE;   // Mandatory
wReq.14 := FALSE;   // Mandatory
wReq.15 := FALSE;   // Mandatory

Status.eComStatus := THIS^.ServiceRequest( wValue := wReq, eCommand := eServiceCommand.SDC_FIXED_RS485MODE, xWrite := TRUE );
END_SET
GET
VAR
	stMode			 : stRS485Mode;
	J				 : INT;
	awSrvAnwser		 : ARRAY [1..2] OF WORD;
	uiParity		 : UINT;
	uiDatabits		 : UINT;
	uiStopbits		 : UINT;
END_VAR
FOR J := 1 TO 2 DO
	Status.eComStatus 		:= THIS^.ServiceRequest( wValue := 16#0000, eCommand := eServiceCommand.SDC_FIXED_RS485MODE, xWrite := FALSE );
	awSrvAnwser[J]			:= MEM.PackBytesToWord(THIS^.abyIntRxBuf[1], THIS^.abyIntRxBuf[0]);
END_FOR

//RS-485 Mode [RW]
//  bit 00..02 - parity - 0: none, 1: even, 2: odd
//  bit 03..04 - data bits: 0: 5, 1: 6, 2: 7, 3: 8
//  bit 05..06 - stop bits: 0: half, 1: one, 2: one and half, 3: two
//  bit 07..15 - RESERVED (write zeros)

uiParity			:= BOOL_TO_UINT(awSrvAnwser[2].0) + BOOL_TO_UINT(awSrvAnwser[2].1) + BOOL_TO_UINT(awSrvAnwser[2].2);
CASE uiParity OF
	eRS485Parity.None			: 	stMode.eParity := eRS485Parity.None;		//0x00								                                    
	eRS485Parity.Even			:  	stMode.eParity := eRS485Parity.Even;		//0x01							                                    
	eRS485Parity.Odd 			:  	stMode.eParity := eRS485Parity.Odd;		//0x02
END_CASE

uiDatabits			:= BOOL_TO_UINT(awSrvAnwser[2].3) + BOOL_TO_UINT(awSrvAnwser[2].4);
CASE uiDatabits OF
	eRS485Databits.Five 		:  	stMode.eDatabits := eRS485Databits.Five;	//0x00
	eRS485Databits.Six 			: 	stMode.eDatabits := eRS485Databits.Six;	//0x01
	eRS485Databits.Seven		:	stMode.eDatabits := eRS485Databits.Seven; //0x02
	eRS485Databits.Eight		: 	stMode.eDatabits := eRS485Databits.Eight; //0x03
END_CASE

uiStopbits			:= BOOL_TO_UINT(awSrvAnwser[2].5) + BOOL_TO_UINT(awSrvAnwser[2].6);
CASE uiStopbits OF
	eRS485Stopbits.Half 		:	stMode.eStopbits := eRS485Stopbits.Half;	//0x00
	eRS485Stopbits.One  		: 	stMode.eStopbits := eRS485Stopbits.One; //0x01
	eRS485Stopbits.OneAndAHalf	: 	stMode.eStopbits := eRS485Stopbits.OneAndAHalf; //0x02
	eRS485Stopbits.Two			: 	stMode.eStopbits := eRS485Stopbits.Two; //0x03
END_CASE

RS485Mode := stMode;

//update classic status
Status.stRS485Mode				:= stMode;
END_GET
END_PROPERTY

/// Please refer to Monarco HAT SPI Protocol Reference Manual for more details!
/// Read/ Write Host Baudrate in steps of 100 Baud.
/// The host side baudrate is configurable by service register 0x012, but it is usually *NOT* needed, as RS-485 side communication parameters are independant on Host side.
///
/// Default communication parameters on Raspberry Pi (Host side) side are; 
/// 	* 115200 Baud, 
/// 	* 8 data bits, no parity, 
///		* 1 stop Bit
///
/// 	* Unit: 100 Bd, Min: 3 (300 Bd), Max 10000 (1 MegaBd)
/// 	12 = 1200 Bd, 
/// 	24 = 2400 Bd, 
/// 	48 = 4800 Bd,
/// 	96 = 9600 Bd,
/// 	192 = 19200 Bd, 
/// 	384 = 38400 Bd,
/// 	576 = 57600 Bd,
/// 	1152 = 115200 Bd
PROPERTY HostBaudrate : UINT
SET
VAR
	uiRate	: UINT;
END_VAR
uiRate := LIMIT( 3, RS485Baudrate, 10000 ); // limit baudrate within accepted range [300 .. 1000000]
Status.eComStatus := THIS^.ServiceRequest( wValue := uiRate, eCommand := eServiceCommand.SDC_FIXED_HOST_UART, xWrite := TRUE );
END_SET
GET
VAR
	J				 : INT;
	awSrvAnwser		 : ARRAY [1..2] OF WORD;
END_VAR
FOR J := 1 TO 2 DO
	Status.eComStatus 		:= THIS^.ServiceRequest( wValue := 16#0000, eCommand := eServiceCommand.SDC_FIXED_HOST_UART, xWrite := FALSE  ) ;
	awSrvAnwser[J]			:= MEM.PackBytesToWord(THIS^.abyIntRxBuf[1], THIS^.abyIntRxBuf[0]);
END_FOR

HostBaudrate 				:= awSrvAnwser[2];

//update classic status
Status.uiRS485Baudrate		:= HostBaudrate;
END_GET
END_PROPERTY

// RS-485 Bytes Received Diagnostics Counter [R]
PROPERTY RS485RxC : UINT
GET
VAR
	J				 : INT;
	awSrvAnwser		 : ARRAY [1..2] OF WORD;
END_VAR
FOR J := 1 TO 2 DO
	Status.eComStatus 		:= THIS^.ServiceRequest( wValue := 16#0000, eCommand := eServiceCommand.SDC_FIXED_RS485_RxC, xWrite := FALSE  ) ;
	awSrvAnwser[J]			:= MEM.PackBytesToWord(THIS^.abyIntRxBuf[1], THIS^.abyIntRxBuf[0]);
END_FOR

RS485RxC 					:= awSrvAnwser[2];

//update classic status
Status.uiRS485Baudrate		:= RS485RxC;
END_GET
END_PROPERTY

// RS-485 Bytes Transmitted Diagnostics Counter [R]
PROPERTY RS485TxC : UINT
GET
VAR
	J				 : INT;
	awSrvAnwser		 : ARRAY [1..2] OF WORD;
END_VAR
FOR J := 1 TO 2 DO
	Status.eComStatus 		:= THIS^.ServiceRequest( wValue := 16#0000, eCommand := eServiceCommand.SDC_FIXED_RS485_TxC, xWrite := FALSE  ) ;
	awSrvAnwser[J]			:= MEM.PackBytesToWord(THIS^.abyIntRxBuf[1], THIS^.abyIntRxBuf[0]);
END_FOR

RS485TxC 					:= awSrvAnwser[2];

//update classic status
Status.uiRS485Baudrate		:= RS485TxC;
END_GET
END_PROPERTY

// RS-485 RX Framing Error Diagnostics Counter [R]
PROPERTY RS485FxC : UINT
GET
VAR
	J				 : INT;
	awSrvAnwser		 : ARRAY [1..2] OF WORD;
END_VAR
FOR J := 1 TO 2 DO
	Status.eComStatus 		:= THIS^.ServiceRequest( wValue := 16#0000, eCommand := eServiceCommand.SDC_FIXED_RS485_FxC, xWrite := FALSE  ) ;
	awSrvAnwser[J]			:= MEM.PackBytesToWord(THIS^.abyIntRxBuf[1], THIS^.abyIntRxBuf[0]);
END_FOR

RS485FxC 					:= awSrvAnwser[2];

//update classic status
Status.uiRS485Baudrate		:= RS485FxC;
END_GET
END_PROPERTY

//RS-485 RX Parity Error Diagnostics Counter [R]
PROPERTY RS485PxC : UINT
GET
VAR
	J				 : INT;
	awSrvAnwser		 : ARRAY [1..2] OF WORD;
END_VAR
FOR J := 1 TO 2 DO
	Status.eComStatus 		:= THIS^.ServiceRequest( wValue := 16#0000, eCommand := eServiceCommand.SDC_FIXED_RS485_PxC, xWrite := FALSE  ) ;
	awSrvAnwser[J]			:= MEM.PackBytesToWord(THIS^.abyIntRxBuf[1], THIS^.abyIntRxBuf[0]);
END_FOR

RS485PxC 					:= awSrvAnwser[2];

//update classic status
Status.uiRS485Baudrate		:= RS485PxC;
END_GET
END_PROPERTY

// Write Digital Out Channels
METHOD setDOut : eMonarcoComStatus;
VAR_INPUT
	stDOut			: stDOut;
END_VAR
THIS^.abyIntTxBuf[7].1	:= stDOut.xDOut1;
THIS^.abyIntTxBuf[7].2	:= stDOut.xDOut2;
THIS^.abyIntTxBuf[7].3	:= stDOut.xDOut3;
THIS^.abyIntTxBuf[7].4	:= stDOut.xDOut4;

//send/receive
setDOut							:= THIS^.dataTransfer();

// update classic status
THIS^.Status.stDOut				:= stDOut;
END_METHOD

//Set a free configurable service request to write or read a service register
METHOD ServiceRequest : eMonarcoComStatus;
VAR_INPUT
	wValue 				: WORD;				/// The value which you want set,
	eCommand 			: eServiceCommand;	/// The service which you want to set,
	xWrite				: BOOL := TRUE;		/// Write = TRUE (default), Read only = FALSE
END_VAR
VAR
	stRequest			: stServiceRequest;	
END_VAR
stRequest.wServiceValue			:= wValue;
stRequest.wServiceAddress		:= Paramlist.SDC_ADDRESS_MASK AND TO_WORD(eCommand);
stRequest.wServiceAddress.12	:= xWrite;
                      	
// Service Data Request     	
THIS^.abyIntTxBuf[0]			:= WORD_TO_BYTE(stRequest.wServiceValue); // ServiceValueHi;
THIS^.abyIntTxBuf[1]			:= WORD_TO_BYTE(SHR(stRequest.wServiceValue,8)); // ServiceValueLo;
THIS^.abyIntTxBuf[2]			:= WORD_TO_BYTE(stRequest.wServiceAddress);//ServiceRegisterHi;
THIS^.abyIntTxBuf[3]			:= WORD_TO_BYTE(SHR(stRequest.wServiceAddress,8));//ServiceRegisterLo;
                            	
//send/receive              	
ServiceRequest 					:= THIS^.dataTransfer();
END_METHOD

/// Reads the Monarco HAT CPU ID of the embedded microcontroller (MCU)
PROPERTY getCpuID : LWORD
GET
getCpuID := THIS^.Status.stHATinfo.lwCpuID;
END_GET
END_PROPERTY

/// Reads the Monarco HAT Firmware Version
PROPERTY getFwVersion : DWORD
GET
GetFwVersion := THIS^.Status.stHATinfo.dwFwVersion;
END_GET
END_PROPERTY

/// reads the Monarco HAT Hardware Revision
PROPERTY getHwVersion : DWORD
GET
GetHwVersion := THIS^.Status.stHATinfo.dwHwVersion;
END_GET
END_PROPERTY

/// Reads the "classic" status via a property
PROPERTY getStatus : stMonarcoStatus
GET
getStatus := THIS^.Status;
END_GET
END_PROPERTY

/// Set the Analog outputs to Current Loop or Voltage
/// Set the RS485 shunt resistor
PROPERTY HWConfig1 : stHWConfig1
SET
VAR
	Cfg1					: stHWConfig1;
	wReq					: WORD;
END_VAR
Cfg1   := HWConfig1;
wReq.0 := Cfg1.xTerminated;
wReq.1 := Cfg1.xAIN1shunt;
wReq.2 := Cfg1.xAIN2shunt;
wReq.3 := FALSE;	// Mandatory
wReq.4 := FALSE;	// Mandatory
wReq.5 := FALSE;	// Mandatory
wReq.6 := FALSE;	// Mandatory
wReq.7 := FALSE;	// Mandatory
wReq.8 := FALSE;	// Mandatory
wReq.9 := FALSE;	// Mandatory
wReq.10 := FALSE;   // Mandatory
wReq.11 := FALSE;   // Mandatory
wReq.12 := FALSE;   // Mandatory
wReq.13 := FALSE;   // Mandatory
wReq.14 := FALSE;   // Mandatory
wReq.15 := FALSE;   // Mandatory

Status.eComStatus := THIS^.ServiceRequest( wValue := wReq, eCommand := eServiceCommand.SDC_FIXED_HWConfig1, xWrite := TRUE );
END_SET
GET
VAR
	J				 : INT;
	awSrvAnwser		 : ARRAY [1..2] OF WORD;
	stCfg1			 : stHWConfig1;
END_VAR
FOR J := 1 TO 2 DO
	Status.eComStatus 		:= THIS^.ServiceRequest( wValue := 16#0000, eCommand := eServiceCommand.SDC_FIXED_HWConfig1, xWrite := FALSE ) ;
	awSrvAnwser[J]			:= MEM.PackBytesToWord(THIS^.abyIntRxBuf[1], THIS^.abyIntRxBuf[0]);
END_FOR

stCfg1.xTerminated			:= awSrvAnwser[2].0;
stCfg1.xAIN1shunt			:= awSrvAnwser[2].1;
stCfg1.xAIN2shunt			:= awSrvAnwser[2].2;

HWConfig1					:= stCfg1;

//update classic status
Status.stHWConfig1			:= HWConfig1;
END_GET
END_PROPERTY

/// Read / Write the Watchdog Timeout
/// Unit: 1 = 1 msec; 0 = watchdog disabled; default = 100msec.
PROPERTY Watchdog : UINT;
SET
Status.eComStatus := THIS^.ServiceRequest( wValue := Watchdog, eCommand := eServiceCommand.SDC_FIXED_WATCHDOG, xWrite := TRUE );
END_SET
GET
VAR
	J				 : INT;
	awSrvAnwser		 : ARRAY [1..2] OF WORD;
END_VAR
FOR J := 1 TO 2 DO
	Status.eComStatus 		:= THIS^.ServiceRequest( wValue := 16#0000, eCommand := eServiceCommand.SDC_FIXED_WATCHDOG, xWrite := FALSE  ) ;
	awSrvAnwser[J]			:= MEM.PackBytesToWord(THIS^.abyIntRxBuf[1], THIS^.abyIntRxBuf[0]);
END_FOR

Watchdog 					:= awSrvAnwser[2];

//update classic status
Status.uiWatchDog			:= Watchdog;
END_GET
END_PROPERTY

/// Reads the most recent service reponse
METHOD getServiceResponse : eMonarcoComStatus;
VAR_OUTPUT
	Response	: stServiceResponse;
END_VAR
VAR	
	rsp			: stServiceResponse;
END_VAR
//send/receive           
getServiceResponse			:= THIS^.dataTransfer();

rsp.wServiceValue			:= MEM.PackBytesToWord(abyIntRxBuf[1],abyIntRxBuf[0]);
rsp.wServiceAddress			:= MEM.PackBytesToWord(abyIntRxBuf[3],abyIntRxBuf[2]);

CASE rsp.wServiceValue OF
	/// Set the error bit
	Paramlist.MONARCO_SERVICE_STATUS_OK			: 	Response.xError		:= FALSE;						
	Paramlist.MONARCO_SERVICE_ERROR_UNKNOWN_REG	: 	Response.xError		:= TRUE;
	Paramlist.MONARCO_SERVICE_ERROR_CRC			: 	Response.xError		:= TRUE;										
END_CASE

/// just give the response back
Response.wServiceValue		:= MEM.PackBytesToWord(abyIntRxBuf[1],abyIntRxBuf[0]);
Response.wServiceAddress	:= MEM.PackBytesToWord(abyIntRxBuf[3],abyIntRxBuf[2]);

// set status
Status.stLastServiceResponse := Response;
END_METHOD

/// Read / write the control byte
PROPERTY ControlByte : stControlByte
SET
VAR
	eComStat	: eMonarcoComStatus;
END_VAR
THIS^.abyIntRxBuf[4].0 := ControlByte.xStatusLEDctrl;
THIS^.abyIntRxBuf[4].1 := ControlByte.xStatusLEDvalue;
THIS^.abyIntRxBuf[4].2 := ControlByte.xOneWireShutdown;
THIS^.abyIntRxBuf[4].3 := FALSE;
THIS^.abyIntRxBuf[4].4 := ControlByte.xCounter1Reset;
THIS^.abyIntRxBuf[4].5 := ControlByte.xCounter2Reset;
THIS^.abyIntRxBuf[4].6 := ControlByte.xSignOfLife0;
THIS^.abyIntRxBuf[4].7 := ControlByte.xSignOfLife1;

//send/receive
THIS^.Status.eComStatus	:= THIS^.dataTransfer();

// update classic status;
THIS^.Status.stControlByte	:=  ControlByte;
END_SET
GET
VAR
	ctrlbyte	:	stControlByte;
END_VAR
//send/receive
THIS^.Status.eComStatus		:= THIS^.dataTransfer();
 					
ctrlbyte.xStatusLEDctrl 	:= abyIntRxBuf[4].0;
ctrlbyte.xStatusLEDvalue 	:= abyIntRxBuf[4].1;
ctrlbyte.xOneWireShutdown	:= abyIntRxBuf[4].2;
ctrlbyte.xReserved	 		:= FALSE;				// Mandatory
ctrlbyte.xCounter1Reset 	:= abyIntRxBuf[4].4;
ctrlbyte.xCounter2Reset 	:= abyIntRxBuf[4].5;
ctrlbyte.xSignOfLife0 		:= abyIntRxBuf[4].6;
ctrlbyte.xSignOfLife1 		:= abyIntRxBuf[4].7;

// return the anwser
ControlByte					:= ctrlbyte;

// update classic status
THIS^.Status.stControlByte	:= ctrlbyte;
END_GET
END_PROPERTY

//  Read the Digital In channel value's
METHOD getDIn : eMonarcoComStatus;
VAR_OUTPUT
	stDIn				: stDIn;
END_VAR
// send/receive
getDIn 							:= THIS^.DataTransfer();

stDIn.xDIn1 					:= THIS^.abyIntRxBuf[7].0;
stDIn.xDIn2						:= THIS^.abyIntRxBuf[7].1;
stDIn.xDIn3						:= THIS^.abyIntRxBuf[7].2;
stDIn.xDIn4						:= THIS^.abyIntRxBuf[7].3;

// update classic status
THIS^.Status.stDIn				:= stDIn;
END_METHOD

// Read the AIn channel value's
METHOD getAIn : eMonarcoComStatus;
VAR_OUTPUT
	AIn				: stAIn;
END_VAR
// send/receive
getAIn 							:= THIS^.DataTransfer();

AIn.wAIn1						:= MEM.PackBytesToWord(THIS^.abyIntRxBuf[21],THIS^.abyIntRxBuf[20]);
AIn.wAIn2						:= MEM.PackBytesToWord(THIS^.abyIntRxBuf[23],THIS^.abyIntRxBuf[22]);

// update classic status
THIS^.Status.stAIn				:= AIn;
END_METHOD

//// Write the raw received anwser, for ease of use the CRC16 will be  automaticly added before sending
METHOD setRawTxBuf : eMonarcoComStatus
VAR_INPUT
	/// SDC [4 bytes]:
	ServiceValueHi   : BYTE; /// Read register request byte1
	ServiceValueLo   : BYTE; /// Read register request byte2
	ServiceRegisterHi: BYTE; /// Read register request byte3
	ServiceRegisterLo: BYTE; /// Read register request byte4
	/// Process data [20 bytes]: 
	ControlByte 	 : BYTE; /// Control byte: status LED mask on, value off
	LEDMask			 : BYTE; /// User LEDs mask
	LEDValue		 : BYTE; /// User LEDs value
	DigitalOuts 	 : BYTE; /// Digital outputs: 0x00 (all off)
	PWM1_F_HiByte 	 : BYTE; /// PWM1 frequency: 0x7D00 = 32000: prescaler = 1, TOP = 32000: frequency = 1000 Hz
	PWM1_F_LoByte 	 : BYTE; /// PWM1 frequency: 0x7D00 = 32000: prescaler = 1, TOP = 32000: frequency = 1000 Hz
	PWM1_ChA_HiByte  : BYTE; /// PWM1 Channel A (DOUT1) duty cycle: 0x0000: PWM disabled
	PWM1_ChA_LoByte  : BYTE; /// PWM1 Channel A (DOUT1) duty cycle: 0x0000: PWM disabled
	PWM1_ChB_HiByte  : BYTE; /// PWM1 Channel B (DOUT2) duty cycle: 0x0000: PWM disabled
	PWM1_ChB_LoByte  : BYTE; /// PWM1 Channel B (DOUT2) duty cycle: 0x0000: PWM disabled
	PWM1_ChC_HiByte  : BYTE; /// PWM1 Channel C (DOUT3) duty cycle: 0x0000: PWM disabled
	PWM1_ChC_LoByte  : BYTE; /// PWM1 Channel C (DOUT3) duty cycle: 0x0000: PWM disabled
	PWM2_F_HiByte 	 : BYTE; /// PWM2 frequency: 0x0C80 = 3200: prescaler = 1, TOP = 3200: frequency = 10000 Hz
	PWM2_F_LoByte 	 : BYTE; /// PWM2 frequency: 0x0C80 = 3200: prescaler = 1, TOP = 3200: frequency = 10000 Hz
	PWM2_ChA_HiByte  : BYTE; /// PWM2 Channel A (DOUT4) duty cycle: 0x0000: PWM disabled
	PWM2_ChA_LoByte  : BYTE; /// PWM2 Channel A (DOUT4) duty cycle: 0x0000: PWM disabled
	AOut1_Hi		 : BYTE; /// Analog output 1: 0x0999 = 2457: 6.0 V
	AOut1_Lo		 : BYTE; /// Analog output 1: 0x0999 = 2457: 6.0 V
	AOut2_Hi		 : BYTE; /// Analog output 2: 0x04CC = 1228: 3.0 V
	AOut2_Lo		 : BYTE; /// Analog output 2: 0x04CC = 1228: 3.0 V
END_VAR
/// Service Data Request (SDC) [4 bytes]
THIS^.abyIntTxBuf[0] 			:= ServiceValueHi;
THIS^.abyIntTxBuf[1] 			:= ServiceValueLo;
THIS^.abyIntTxBuf[2] 			:= ServiceRegisterHi;
THIS^.abyIntTxBuf[3] 			:= ServiceRegisterLo;
THIS^.abyIntTxBuf[4] 			:= ControlByte; 
THIS^.abyIntTxBuf[5] 			:= LEDMask; 
THIS^.abyIntTxBuf[6] 			:= LEDValue; 
THIS^.abyIntTxBuf[7] 			:= DigitalOuts; 
THIS^.abyIntTxBuf[8] 			:= PWM1_F_HiByte; 
THIS^.abyIntTxBuf[9] 			:= PWM1_F_LoByte; 
THIS^.abyIntTxBuf[10] 			:= PWM1_ChA_HiByte; 
THIS^.abyIntTxBuf[11] 			:= PWM1_ChA_LoByte;
THIS^.abyIntTxBuf[12] 			:= PWM1_ChB_HiByte; 
THIS^.abyIntTxBuf[13] 			:= PWM1_ChB_LoByte; 
THIS^.abyIntTxBuf[14] 			:= PWM1_ChC_HiByte; 
THIS^.abyIntTxBuf[15] 			:= PWM1_ChC_LoByte;
THIS^.abyIntTxBuf[16] 			:= PWM2_F_HiByte;
THIS^.abyIntTxBuf[17] 			:= PWM2_F_LoByte;
THIS^.abyIntTxBuf[18] 			:= PWM2_ChA_HiByte;
THIS^.abyIntTxBuf[19] 			:= PWM2_ChA_LoByte;
THIS^.abyIntTxBuf[20] 			:= AOut1_Hi;
THIS^.abyIntTxBuf[21] 			:= AOut1_Lo;
THIS^.abyIntTxBuf[22] 			:= AOut2_Hi;
THIS^.abyIntTxBuf[23] 			:= AOut2_Lo;

//send/receive
setRawTxBuf 					:= THIS^.dataTransfer();
END_METHOD

/// Read the raw received anwser
METHOD getRawRxBuf :  ARRAY [0..(ParamList.MONARCO_STRUCT_SIZE-1)] OF BYTE;
getRawRxBuf := THIS^.abyIntRxBuf;

//update classic status
THIS^.status.abyRawRxBuffer := getRawRxBuf;
END_METHOD

/// Write Analog Out Channels
METHOD setAOut : eMonarcoComStatus;
VAR_INPUT
	stAOut				: stAOut;			
END_VAR
VAR	
	v1					: WORD;
	v2					: WORD;
END_VAR
// limit the value's
v1 := LIMIT(0, stAOut.wAOut1, Paramlist.MONARCO_ADC_RANGE_MAX );
v2 := LIMIT(0, stAOut.wAOut2, Paramlist.MONARCO_ADC_RANGE_MAX );

THIS^.abyIntTxBuf[20] 			:= WORD_TO_BYTE(v1);
THIS^.abyIntTxBuf[21] 			:= WORD_TO_BYTE(SHR(v1,8));
THIS^.abyIntTxBuf[22] 			:= WORD_TO_BYTE(v2);       
THIS^.abyIntTxBuf[23] 			:= WORD_TO_BYTE(SHR(v2,8));

//send/receive
setAOut 						:= THIS^.dataTransfer();

// update classic status
THIS^.Status.stAOut				:= stAOut;
END_METHOD

// Get / Set configure COUNTER1
PROPERTY Counter1Config : stCounter1Config
SET
VAR
	stConfig				: stCounter1Config;
	wReq					: WORD;
END_VAR
/// COUNTER1 Configuration;
///   Mode;
///	   * Off,
///    * Pulse counting,
///    * Quadrature encoder,
///   Direction (only for pulse counting mode):
///     * Up
///     * [FUTURE] external control, low/high = up/down
///   Active Edge (only for pulse counting mode):
///     * Rising
///     * Falling
///     * Both
stConfig   := Counter1Config;
CASE stConfig.eMode OF
	eCounterMode.Off					: 	wReq.0 := FALSE;	//0x00
											wReq.1 := FALSE;
											wReq.2 := FALSE;
										
	eCounterMode.PulseCounting			:  	wReq.0 := TRUE;		//0x01
											wReq.1 := FALSE;
											wReq.2 := FALSE;
										
	eCounterMode.QuadratureEncoder 		:  	wReq.0 := FALSE;	//0x02
											wReq.1 := TRUE;
											wReq.2 := FALSE;
END_CASE

CASE stConfig.eDirection OF
	eCounterDirection.up				:  	wReq.3 := FALSE;	//0x00
											wReq.4 := FALSE;
											wReq.5 := FALSE;
									
	eCounterDirection.External_Control1	: 	wReq.3 := TRUE;		//0x01	[FUTURE] external control, low/high = up/down
											wReq.4 := FALSE;
											wReq.5 := FALSE;
END_CASE

CASE stConfig.eActiveEdge OF
	eCounterActiveEdge.rising 			:	wReq.6 := FALSE;	//0x00
											wReq.7 := FALSE;
											
	eCounterActiveEdge.falling 			: 	wReq.6 := TRUE;		//0x01
											wReq.7 := FALSE;
											
	eCounterActiveEdge.both				: 	wReq.6 := FALSE;	//0x02
											wReq.7 := TRUE;							
END_CASE

wReq.8 := FALSE;	// Mandatory
wReq.9 := FALSE;	// Mandatory
wReq.10 := FALSE;   // Mandatory
wReq.11 := FALSE;   // Mandatory
wReq.12 := FALSE;   // Mandatory
wReq.13 := FALSE;   // Mandatory
wReq.14 := FALSE;   // Mandatory
wReq.15 := FALSE;   // Mandatory

Status.eComStatus := THIS^.ServiceRequest( wValue := wReq, eCommand := eServiceCommand.SDC_FIXED_CNT1MODE, xWrite := TRUE );

// update classic status;
THIS^.Status.stCounter1Config := stConfig;
END_SET
GET
VAR
	stConfig		: stCounter1Config;
	J				: INT;
	awSrvAnwser		: ARRAY [1..2] OF WORD;
	uiMode		 	: UINT;
	uiDirection		: UINT;
	uiActiveEdge	: UINT;
END_VAR
FOR J := 1 TO 2 DO
	Status.eComStatus := THIS^.ServiceRequest( wValue := 16#0000, eCommand := eServiceCommand.SDC_FIXED_CNT1MODE, xWrite := FALSE );
	awSrvAnwser[J]	 := MEM.PackBytesToWord(THIS^.abyIntRxBuf[1], THIS^.abyIntRxBuf[0]);
END_FOR

/// COUNTER1 Configuration;
///   Mode;
///	   * Off,
///    * Pulse counting,
///    * Quadrature encoder,
///   Direction (only for pulse counting mode):
///     * Up
///     * [FUTURE] external control, low/high = up/down
///   Active Edge (only for pulse counting mode):
///     * Rising
///     * Falling
///     * Both

uiMode := BOOL_TO_UINT(awSrvAnwser[2].0) + BOOL_TO_UINT(awSrvAnwser[2].1) + BOOL_TO_UINT(awSrvAnwser[2].2);
CASE uiMode OF
	eCounterMode.Off					: stConfig.eMode := eCounterMode.Off;				//0x00								                                    
	eCounterMode.PulseCounting			: stConfig.eMode := eCounterMode.PulseCounting;		//0x01							                                    
	eCounterMode.QuadratureEncoder		: stConfig.eMode := eCounterMode.QuadratureEncoder;	//0x02
ELSE
	// Weird value returns?
	stConfig.eMode := eCounterMode.Off;
END_CASE

uiDirection	:= BOOL_TO_UINT(awSrvAnwser[2].3) + BOOL_TO_UINT(awSrvAnwser[2].4) + BOOL_TO_UINT(awSrvAnwser[2].5);
CASE uiDirection OF
	eCounterDirection.Up 				: stConfig.eDirection := eCounterDirection.Up;					//0x00
	eCounterDirection.External_Control1	: stConfig.eDirection := eCounterDirection.External_Control1;	//0x01
ELSE
	// [FUTURE] or weird value's?
	stConfig.eDirection := eCounterDirection.External_Control1;
END_CASE

uiActiveEdge :=  BOOL_TO_UINT(awSrvAnwser[2].6) + BOOL_TO_UINT(awSrvAnwser[2].7);
CASE uiActiveEdge OF
	eCounterActiveEdge.Rising 			: stConfig.eActiveEdge := eCounterActiveEdge.Rising;	//0x00
	eCounterActiveEdge.Falling  		: stConfig.eActiveEdge := eCounterActiveEdge.Falling; 	//0x01
	eCounterActiveEdge.Both				: stConfig.eActiveEdge := eCounterActiveEdge.Both; 		//0x02
ELSE
	// Weird value returns?
	stConfig.eActiveEdge := eCounterActiveEdge.Rising;	//0x00		
END_CASE

Counter1Config := stConfig;

//update classic status
Status.stCounter1Config					:= stConfig;
END_GET
END_PROPERTY

// Get / Set configure COUNTER2
PROPERTY Counter2Config : stCounter2Config
SET
VAR
	stConfig				: stCounter2Config;
	wReq					: WORD;
END_VAR
/// COUNTER1 Configuration;
///   Mode;
///	   * Off,
///    * Pulse counting,
///    * Quadrature encoder,
///   Direction (only for pulse counting mode):
///     * Up
///     * [FUTURE] external control, low/high = up/down
///   Active Edge (only for pulse counting mode):
///     * Rising
///     * Falling
///     * Both
///   CAPTURE function active edge:
///     * Disabled
///     * [FUTURE] rising
///     * [FUTURE] falling
///     * [FUTURE] both

stConfig   := Counter2Config;
CASE stConfig.Mode OF
	eCounterMode.Off					: 	wReq.0 := FALSE;	//0x00
											wReq.1 := FALSE;
											wReq.2 := FALSE;
										
	eCounterMode.PulseCounting			:  	wReq.0 := TRUE;		//0x01
											wReq.1 := FALSE;
											wReq.2 := FALSE;
										
	eCounterMode.QuadratureEncoder 		:  	wReq.0 := FALSE;	//0x02
											wReq.1 := TRUE;
											wReq.2 := FALSE;
END_CASE

CASE stConfig.Direction OF
	eCounterDirection.up				:  	wReq.3 := FALSE;	//0x00
											wReq.4 := FALSE;
											wReq.5 := FALSE;
									
	eCounterDirection.External_Control1	: 	wReq.3 := TRUE;		//0x01	[FUTURE] external control, low/high = up/down
											wReq.4 := FALSE;
											wReq.5 := FALSE;
END_CASE

CASE stConfig.ActiveEdge OF
	eCounterActiveEdge.rising 			:	wReq.6 := FALSE;	//0x00
											wReq.7 := FALSE;
											
	eCounterActiveEdge.falling 			: 	wReq.6 := TRUE;		//0x01
											wReq.7 := FALSE;
											
	eCounterActiveEdge.both				: 	wReq.6 := FALSE;	//0x02
											wReq.7 := TRUE;							
END_CASE

CASE stConfig.Capture OF
	eCounterCapture.Disabled 			:	wReq.8 := FALSE;	//0x00
											wReq.9 := FALSE;
											
	eCounterCapture.Rising	 			: 	wReq.8 := TRUE;		//0x01 [FUTURE]
											wReq.9 := FALSE;
											
	eCounterCapture.Falling				: 	wReq.8 := FALSE;	//0x02 [FUTURE]
											wReq.9 := TRUE;		
											
	eCounterCapture.Both				: 	wReq.8 := TRUE;		//0x03 [FUTURE]
											wReq.9 := TRUE;							
END_CASE

wReq.10 := FALSE;   // Mandatory
wReq.11 := FALSE;   // Mandatory
wReq.12 := FALSE;   // Mandatory
wReq.13 := FALSE;   // Mandatory
wReq.14 := FALSE;   // Mandatory
wReq.15 := FALSE;   // Mandatory

Status.eComStatus := THIS^.ServiceRequest( wValue := wReq, eCommand := eServiceCommand.SDC_FIXED_CNT2MODE, xWrite := TRUE );

// update classic status;
THIS^.Status.stCounter2Config := stConfig;
END_SET
GET
VAR
	stConfig		: stCounter2Config;
	J				: INT;
	awSrvAnwser		: ARRAY [1..2] OF WORD;
	uiMode		 	: UINT;
	uiDirection		: UINT;
	uiActiveEdge	: UINT;
	uiCapture		: UINT;
END_VAR
FOR J := 1 TO 2 DO
	Status.eComStatus := THIS^.ServiceRequest( wValue := 16#0000, eCommand := eServiceCommand.SDC_FIXED_CNT2MODE, xWrite := FALSE );
	awSrvAnwser[J]	 := MEM.PackBytesToWord(THIS^.abyIntRxBuf[1], THIS^.abyIntRxBuf[0]);
END_FOR

/// COUNTER2 Configuration;
///   Mode;
///	   * Off,
///    * Pulse counting,
///    * Quadrature encoder,
///   Direction (only for pulse counting mode):
///     * Up
///     * [FUTURE] external control, low/high = up/down
///   Active Edge (only for pulse counting mode):
///     * Rising
///     * Falling
///     * Both
///   CAPTURE function active edge:
///     * Disabled
///     * [FUTURE] rising
///     * [FUTURE] falling
///     * [FUTURE] both

uiMode := BOOL_TO_UINT(awSrvAnwser[2].0) + BOOL_TO_UINT(awSrvAnwser[2].1) + BOOL_TO_UINT(awSrvAnwser[2].2);
CASE uiMode OF
	eCounterMode.Off					: stConfig.Mode := eCounterMode.Off;				//0x00								                                    
	eCounterMode.PulseCounting			: stConfig.Mode := eCounterMode.PulseCounting;		//0x01							                                    
	eCounterMode.QuadratureEncoder		: stConfig.Mode := eCounterMode.QuadratureEncoder;	//0x02
ELSE
	// Weird value returns?
	stConfig.Mode := eCounterMode.Off;
END_CASE

uiDirection	:= BOOL_TO_UINT(awSrvAnwser[2].3) + BOOL_TO_UINT(awSrvAnwser[2].4) + BOOL_TO_UINT(awSrvAnwser[2].5);
CASE uiDirection OF
	eCounterDirection.Up 				: stConfig.Direction := eCounterDirection.Up;					//0x00
	eCounterDirection.External_Control1	: stConfig.Direction := eCounterDirection.External_Control1;	//0x01
ELSE
	// [FUTURE] or weird value's?
	stConfig.Direction := eCounterDirection.External_Control1;
END_CASE

uiActiveEdge :=  BOOL_TO_UINT(awSrvAnwser[2].6) + BOOL_TO_UINT(awSrvAnwser[2].7);
CASE uiActiveEdge OF
	eCounterActiveEdge.Rising 			: stConfig.ActiveEdge := eCounterActiveEdge.Rising;	 //0x00
	eCounterActiveEdge.Falling  		: stConfig.ActiveEdge := eCounterActiveEdge.Falling; //0x01
	eCounterActiveEdge.Both				: stConfig.ActiveEdge := eCounterActiveEdge.Both;    //0x02
ELSE
	// Weird value returns?
	stConfig.ActiveEdge := eCounterActiveEdge.Rising;	//0x00		
END_CASE


uiCapture :=  BOOL_TO_UINT(awSrvAnwser[2].8) + BOOL_TO_UINT(awSrvAnwser[2].9);
CASE uiCapture OF
	eCounterCapture.Disabled 			: stConfig.Capture := eCounterCapture.Disabled;	//0x00
	eCounterCapture.Rising  			: stConfig.Capture := eCounterCapture.Rising; 	//0x01
	eCounterCapture.Falling				: stConfig.Capture := eCounterCapture.Falling; 	//0x02
	eCounterCapture.Both				: stConfig.Capture := eCounterCapture.Both; 	//0x02
ELSE
	// Weird value returns?
	stConfig.Capture := eCounterCapture.Disabled;	//0x00		
END_CASE

Counter2Config := stConfig;

//update classic status
Status.stCounter2Config					:= stConfig;
END_GET
END_PROPERTY

///
///	Just set a frequency between 1 and 100 kHz and the PWM will be set according to below settings;
///
///  f_PWM = 32 MHz / ( prescaler × TOP )
///
/// Where **prescaler can be (1, 8, 64, 512)** and **TOP can be 0 to 65532**.
/// TOP is represented by 14bit value in process data and then multiplied by 4.
/// Modulated value is represented by 16 bits in process data and internally scaled to 0 to TOP range.
/// The lowest possible prescaler should be preferred for given frequency.
/// Because this leads to a bigger value of TOP and so a better resolution of the modulated value.
///
///	==========  ================================  =================================
/// Prescaler   Recommended range low boundary    Recommended range high boundary
///	==========  ================================  =================================
///	1  		    ≥ 1 kHz TOP = 32000               ≤ 100 kHz TOP = 320
///	8           ≥ 100 Hz TOP = 40000              < 1 kHz TOP = 4000
///	64          ≥ 10 Hz TOP = 50000               < 100 Hz TOP = 5000
///	512         ≥ 1 Hz TOP = 62500                < 10 Hz TOP = 6250
///	==========  ================================  =================================
///
/// Example:
///  f_PWM = 10Hz => 16#C352 = 50002
///   prescaler = 64, TOP = 50000 => 10 = 32x10^6 / (64 x 50000)
///
METHOD setPWM1freq : eMonarcoComStatus;
VAR_INPUT
	/// base frequency of the PWM, anywhere from 1Hz to 100kHz (10 Hz = 10, 100kHz = 100000)
	/// A setting higher then 100kHz and lower then 1Hz will be limited to 100kHz and 1Hz.
	udiHz			: UDINT;		
END_VAR
VAR
	_uidiHz			: UDINT;
	ePrescale		: ePrescaler; 	/// Determined prefered prescaler
	uiRangeLow		: UINT;
	uiRangeHigh		: UINT;
	uiTOP			: UINT;			/// Determined TOP setting
	fPWM			: WORD;			
END_VAR
/// clip the input Hz on lower and upper bound, so;
_uidiHz := LIMIT( 1, udiHz, 100000);

/// Determine prescaler and TOP according to table
CASE _uidiHz OF
	1..9			: ePrescale 	:= ePrescaler.ScaleFactor512;
					  uiTOP			:= TO_UINT( (32000000/ 512/ _uidiHz));// interpolate between 1 and 9Hz
	
	10..99			: ePrescale 	:= ePrescaler.ScaleFactor64;
					  uiTOP			:= TO_UINT( (32000000/ 64/ _uidiHz)); // interpolate between 10 and 100Hz
	
	100..999		: ePrescale 	:= ePrescaler.ScaleFactor8;
					  uiTOP			:= TO_UINT( (32000000/ 8/ _uidiHz));// interpolate between 100 and 1000Hz
		
	1000..100000	: ePrescale 	:= ePrescaler.ScaleFactor1;
					  uiTOP			:= TO_UINT( (32000000/ 1/ _uidiHz));// interpolate between 1000 and 100000Hz
END_CASE

/// Now set prescaler
CASE ePrescale OF 
///  00  0 : prescaler =   1
	ePrescaler.ScaleFactor1	: 	fPWM.0 := FALSE;
								fPWM.1 := FALSE;
///  01  1 : prescaler =   8
	ePrescaler.ScaleFactor8 :  	fPWM.0 := TRUE;
								fPWM.1 := FALSE;
///  10  2 : prescaler =  64	
	ePrescaler.ScaleFactor64 :  fPWM.0 := FALSE;
								fPWM.1 := TRUE;
///  11  3 : prescaler = 512	
	ePrescaler.ScaleFactor512 : fPWM.0 := TRUE;
								fPWM.1 := TRUE;
END_CASE

//   8.0   2.0  PWM1 frequency
THIS^.abyIntTxBuf[8] 			:= WORD_TO_BYTE(fPWM) AND 16#FC;	// bitmask to protect prescaler
THIS^.abyIntTxBuf[9] 			:= WORD_TO_BYTE(SHR(fPWM,8));

//send/receive
setPWM1freq 					:= THIS^.dataTransfer();

//// update classic status
THIS^.Status.stPWM1.Freq		:= udiHz;
END_METHOD

///
///	Just set a frequency between 1 and 100 kHz and the PWM will be set according to below settings;
///
///  f_PWM = 32 MHz / ( prescaler × TOP )
///
/// Where **prescaler can be (1, 8, 64, 512)** and **TOP can be 0 to 65532**.
/// TOP is represented by 14bit value in process data and then multiplied by 4.
/// Modulated value is represented by 16 bits in process data and internally scaled to 0 to TOP range.
/// The lowest possible prescaler should be preferred for given frequency.
/// Because this leads to a bigger value of TOP and so a better resolution of the modulated value.
///
///	==========  ================================  =================================
/// Prescaler   Recommended range low boundary    Recommended range high boundary
///	==========  ================================  =================================
///	1  		    ≥ 1 kHz TOP = 32000               ≤ 100 kHz TOP = 320
///	8           ≥ 100 Hz TOP = 40000              < 1 kHz TOP = 4000
///	64          ≥ 10 Hz TOP = 50000               < 100 Hz TOP = 5000
///	512         ≥ 1 Hz TOP = 62500                < 10 Hz TOP = 6250
///	==========  ================================  =================================
///
/// Example:
///  f_PWM = 10Hz => 16#C352 = 50002
///   prescaler = 64, TOP = 50000 => 10 = 32x10^6 / (64 x 50000)
///
METHOD setPWM2freq : eMonarcoComStatus;
VAR_INPUT
	/// base frequency of the PWM, anywhere from 1Hz to 100kHz (10 Hz = 10, 100kHz = 100000)
	/// A setting higher then 100kHz and lower then 1Hz will be limited to 100kHz and 1Hz.
	udiHz			: UDINT;		
END_VAR
VAR
	_uidiHz			: UDINT;
	ePrescale		: ePrescaler; 	/// Determined prefered prescaler
	uiRangeLow		: UINT;
	uiRangeHigh		: UINT;
	uiTOP			: UINT;			/// Determined TOP setting
	fPWM			: WORD;			
END_VAR
/// clip the input Hz on lower and upper bound;
_uidiHz := LIMIT( 1, udiHz, 100000);

//// Determine prescaler and TOP according to table
CASE _uidiHz OF
	1..9			: ePrescale 	:= ePrescaler.ScaleFactor512;
					  uiTOP			:= TO_UINT( (32000000/ 512/ _uidiHz));// interpolate between 1 and 9Hz
	
	10..99			: ePrescale 	:= ePrescaler.ScaleFactor64;
					  uiTOP			:= TO_UINT( (32000000/ 64/ _uidiHz)); // interpolate between 10 and 100Hz
	
	100..999		: ePrescale 	:= ePrescaler.ScaleFactor8;
					  uiTOP			:= TO_UINT( (32000000/ 8/ _uidiHz));// interpolate between 100 and 1000Hz
		
	1000..100000	: ePrescale 	:= ePrescaler.ScaleFactor1;
					  uiTOP			:= TO_UINT( (32000000/ 1/ _uidiHz));// interpolate between 1000 and 100000Hz
END_CASE

/// Now set prescaler
/// bit 15 ..  2 : TOP / 4
CASE ePrescale OF 
///  00  0 : prescaler =   1
	ePrescaler.ScaleFactor1	: 	fPWM.0 := FALSE;
								fPWM.1 := FALSE;
///  01  1 : prescaler =   8
	ePrescaler.ScaleFactor8 :  	fPWM.0 := TRUE;
								fPWM.1 := FALSE;
///  10  2 : prescaler =  64	
	ePrescaler.ScaleFactor64 :  fPWM.0 := FALSE;
								fPWM.1 := TRUE;
///  11  3 : prescaler = 512	
	ePrescaler.ScaleFactor512 : fPWM.0 := TRUE;
								fPWM.1 := TRUE;
END_CASE

//   8.0   2.0  PWM1 frequency
THIS^.abyIntTxBuf[16] 			:= WORD_TO_BYTE(fPWM);
THIS^.abyIntTxBuf[17] 			:= WORD_TO_BYTE(SHR(fPWM,8));

//send/receive
setPWM2freq 					:= THIS^.dataTransfer();

//// update classic status
THIS^.Status.stPWM2.Freq 		:= udiHz;
END_METHOD

/// Set PWM1 Channel A (DOUT1) duty cycle   
METHOD setDutyCycleDOut1 : eMonarcoComStatus
VAR_INPUT
	/// Duty Cycle [0.0 .. 1.0] with 0 = 0% and 1 = 100%
	rDutyCycle			: REAL;
END_VAR
VAR
	/// Duty Cycle as a Word (0..65535)
	wDC			: WORD;
END_VAR
wDC := getDC( rDutyCycle := rDutyCycle );

//   10.0   2.0  PWM1 Dutycycle ch A
THIS^.abyIntTxBuf[10] 				:= WORD_TO_BYTE(wDC);	// bitmask to protect prescaler
THIS^.abyIntTxBuf[11] 				:= WORD_TO_BYTE(SHR(wDC,8));

//send/receive
setDutyCycleDOut1 					:= THIS^.dataTransfer();

//// update classic status
THIS^.Status.stPWM1.DutyCycleDOut1	:= wDC;
END_METHOD

// Set PWM1 Channel B (DOUT2) duty cycle   
METHOD setDutyCycleDOut2 : eMonarcoComStatus
VAR_INPUT
	// Duty Cycle [0.0 .. 1.0] with 0 = 0% and 1 = 100%
	rDutyCycle			: REAL;
END_VAR
VAR
	/// Duty Cycle as a Word (0..65535)
	wDC			: WORD;
END_VAR
wDC := getDC( rDutyCycle := rDutyCycle );

//   12.0   2.0  PWM1 Dutycycle ch B
THIS^.abyIntTxBuf[12] 				:= WORD_TO_BYTE(wDC);	// bitmask to protect prescaler
THIS^.abyIntTxBuf[13] 				:= WORD_TO_BYTE(SHR(wDC,8));

//send/receive
setDutyCycleDOut2 					:= THIS^.dataTransfer();

//// update classic status
THIS^.Status.stPWM1.DutyCycleDOut2	:= wDC;
END_METHOD

// Set PWM1 Channel C (DOUT3) duty cycle   
METHOD setDutyCycleDOut3 : eMonarcoComStatus
VAR_INPUT
	// Duty Cycle [0.0 .. 1.0] with 0 = 0% and 1 = 100%
	rDutyCycle			: REAL;
END_VAR
VAR
	/// Duty Cycle as a Word (0..65535)
	wDC			: WORD;
END_VAR
wDC := getDC( rDutyCycle := rDutyCycle );

//   12.0   2.0  PWM1 Dutycycle ch C
THIS^.abyIntTxBuf[14] 				:= WORD_TO_BYTE(wDC);	// bitmask to protect prescaler
THIS^.abyIntTxBuf[15] 				:= WORD_TO_BYTE(SHR(wDC,8));

//send/receive
setDutyCycleDOut3 					:= THIS^.dataTransfer();

//// update classic status
THIS^.Status.stPWM1.DutyCycleDOut3	:= wDC;
END_METHOD

// Set PWM1 Channel B (DOUT2) duty cycle   
METHOD setDutyCycleDOut4 : eMonarcoComStatus
VAR_INPUT
	// Duty Cycle [0.0 .. 1.0] with 0 = 0% and 1 = 100%
	rDutyCycle			: REAL;
END_VAR
VAR
	/// Duty Cycle as a Word (0..65535)
	wDC			: WORD;
END_VAR
wDC := getDC( rDutyCycle := rDutyCycle );

//   18.0   2.0  PWM2 Dutycycle ch A
THIS^.abyIntTxBuf[18] 				:= WORD_TO_BYTE(wDC);	// bitmask to protect prescaler
THIS^.abyIntTxBuf[19] 				:= WORD_TO_BYTE(SHR(wDC,8));

//send/receive
setDutyCycleDOut4 					:= THIS^.dataTransfer();

//// update classic status
THIS^.Status.stPWM2.DutyCycleDOut4	:= wDC;
END_METHOD

///   Set User LEDs (0..7) On / Off
METHOD SetUserLED : eMonarcoComStatus
VAR_INPUT
	/// Sets Userled 1..8 on or off
	byLeds		:	BYTE;
END_VAR
//   10.0   2.0  PWM1 Dutycycle ch A
THIS^.abyIntTxBuf[5] 				:= byLeds;	// set userled mask
THIS^.abyIntTxBuf[6] 				:= byLeds;	// set userled

//send/receive
SetUserLED 							:= THIS^.dataTransfer();

//// update classic status
THIS^.Status.byUserLeds				:= byLeds;
END_METHOD

END_FUNCTION_BLOCK

// Functions/getDC
/// Transforms a factor (0.00 to 1.00) to a Word 0..65535)
FUNCTION getDC : WORD
VAR_INPUT
	rDutyCycle	: REAL;
END_VAR

IF rDutyCycle <= 0 THEN
	getDC := TO_WORD(0);
ELSIF rDutyCycle > 1 THEN
 	getDC := TO_WORD(65535);
ELSE
	getDC := TO_WORD( TO_REAL(65536-16)/(100-0) * rDutyCycle );
END_IF;

END_FUNCTION

// Library Information/GetLibVersionNumber
// This function has been automatically generated from the project information.
FUNCTION GetLibVersionNumber : DWORD
VAR_INPUT
	
END_VAR

GetLibVersionNumber := 589827;

END_FUNCTION

// Library Information/GetLibVersion
// This function has been automatically generated from the project information.
FUNCTION GetLibVersion : VERSION
VAR_INPUT
	
END_VAR

GetLibVersion.uiMajor := 0;
GetLibVersion.uiMinor := 9;
GetLibVersion.uiServicePack := 0;
GetLibVersion.uiPatch := 3;

END_FUNCTION

// Library Information/IsLibReleased
// This function has been automatically generated from the project information.
FUNCTION IsLibReleased : BOOL
VAR_INPUT
	
END_VAR

IsLibReleased := FALSE;

END_FUNCTION
